(* IEC 61131-3 sources: s22-soft-shell/st_interpret/tests/test_inputs/execution/st_subset_8-9, 9 files *)

(* ---- counterinoutfunction.st ---- *)
// This function is designed to test IN_OUT variable.
// Takes in_out integer and adds 1 to it "counting up by 1"
// Then returns new count  with variable instead of function name
// function name returns true to indicate success
FUNCTION CounterInOutFunction : BOOL //BOOL is the return parameter data type
VAR_IN_OUT
  InOut1 :	INT; //IN_OUT parameter
END_VAR

  InOut1 := InOut1 + 1;

  CounterFunction:= 'TRUE'; //Set the return parameter

END_FUNCTION

(* ---- counteroutputfunction.st ---- *)
// This function is designed to test Output variable.
// Takes input integer and adds 1 to it "counting up by 1"
// Then returns new count using Output variable instead of function name
// function name returns true to indicate success
FUNCTION CounterOutputFunction : BOOL //BOOL is the return parameter data type
VAR_INPUT
  Input1 :	INT; //Input parameter
END_VAR
VAR_OUTPUT
  Output1 :	INT; //Output parameter
END_VAR

  Output1 := Input1 + 1;

  CounterFunction:= 'TRUE'; //Set the return parameter

END_FUNCTION

(* ---- simpleaddfunction.st ---- *)
FUNCTION SimpleAddFunction : INT //INT is the return parameter data type
VAR_INPUT
  Input1 :	INT; //Input parameter 1 to the function
  Input2 :	INT; //Input parameter 2 to the function
END_VAR

VAR
  Sum :	INT; //Local variable for temporary calculation
END_VAR

  Sum:= Input1 + Input2; //Total sum

  SimpleAddFunction:= Sum; //Set the return parameter

END_FUNCTION

(* ---- threevarfunction.st ---- *)
// This function is designed to test Output variable.
// Takes input integer and adds 1 to it "counting up by 1"
// Then returns new count using Output variable instead of function name
// function name returns true to indicate success
FUNCTION ThreeVarFunction : BOOL //BOOL is the return parameter data type
VAR_INPUT
  Input1 :	INT; //Input parameter
END_VAR
VAR_OUTPUT
  Output1 :	INT; //Output parameter
END_VAR
VAR_OUTPUT
  InOut1 :	INT; //Output parameter
END_VAR

  Output1 := Input1 + 1;

  InOut1  := InOut1 + 2;

  CounterFunction:= 'TRUE'; //Set the return parameter

END_FUNCTION

(* ---- valueaveragefunction.st ---- *)
FUNCTION ValueAverageFunction : REAL //REAL is the return parameter data type
VAR_INPUT
  Value1 :	REAL; //Input parameter 1 to the function
  Value2 :	REAL; //Input parameter 2 to the function
END_VAR

VAR
  Sum :	REAL; //Local variable for temporary calculation
END_VAR

  Sum:= Value1 + Value2; //Total sum
  Sum:= Sum/2; //Average

  ValueAverageFunction := Sum; //Set the return parameter

END_FUNCTION

(* ---- 09_Main_Add.st ---- *)
//Testing simple function call to add two numbers together
PROGRAM 09_Main_Add
    VAR
	a : int;
        b : int;
        result0 : int;
        result1 : int;
        result2 : int;
        result3 : int;
        ST_TESTING_RESULT : bool;
    END_VAR
        a := 3;
        b := 5;

        // four different ways of function input
        result0 := SimpleAddFunction(10, 10+5); // expects outputs of 25

        result1 := SimpleAddFunction(Input1 := 5, Input2 := 10);// expects outputs of 15

        result2 := SimpleAddFunction(a, b); // expects outputs of 8

        result3 := SimpleAddFunction(Input1 := a, Input2 := b); // expects outputs of 8

        ST_TESTING_RESULT := (result0 = 25 & result1 = 15) & (result2 = 8 & result3 = 8);

END_PROGRAM

(* ---- 09_Main_Avg.st ---- *)
//Testing simple function call to get average of two numbers
PROGRAM 09_Main_Avg
    VAR
	a : real;
        b : real;
        avg1 : real;
        avg2 : real;
        avg3 : real;
        avg4 : real;
        ST_TESTING_RESULT : bool;
    END_VAR
        a := 4;
        b := 6;

        // four different ways of function input
        avg1 := ValueAverageFunction(10, 10+5); // expects 12.5

        avg2 := ValueAverageFunction(Value1 := 5, Value2 := 10); // expects 7.5

        avg3 := ValueAverageFunction(a, b); // expects 5

        avg4 := ValueAverageFunction(Value1 := a, Value2 := b); // expects 5

        ST_TESTING_RESULT := (avg1 = 12.5 & avg2 = 7.5) & (avg3 = 5.0 & avg4 = 5.0);

END_PROGRAM

(* ---- 09_Main_Context_Check.st ---- *)
//Testing to insure seperation of context, Input2 and Sum variables being used in main and add function
PROGRAM 09_Main_Context_Check
    VAR
	    a : int;
        b : int;
        Input2 : int;
        Sum : INT;
        result0 : int;
        result1 : int;
        ST_TESTING_RESULT : bool;
    END_VAR
        a := 3;
        b := 5;
        Input2 := 10;
        Sum := 2;

        result0 := SimpleAddFunction(a, b); // expects outputs of 8

        result1 := SimpleAddFunction(Input1 := a, Input2 := b); // expects outputs of 8

        ST_TESTING_RESULT := (result0 = 8 & result1 = 8) & (Input2 = 10 & Sum = 2);

END_PROGRAM

(* ---- 09_Main_Demo_01.st ---- *)
// Testing for GO West Example use case example
// program doesnt go into while loop without C API
// is used to set INPUT1 or INPUT2 to TRUE
// x represents number of loops INPUT1 and INPUT2 are both true during
// OUTPUT1 represents number of loops
PROGRAM 09_Main_Demo_01
    VAR
	x : int;
        INPUT1 : bool;
        INPUT2 : bool;
        OUTPUT1 : int;
        ST_TESTING_RESULT : bool;
    END_VAR
        x := 0;
        INPUT1 := False;
        INPUT2 := False ;
        OUTPUT1 := 0 ;
//API would control INPUTs after here HERE here

        WHILE (INPUT1) OR (INPUT2) DO
            If (INPUT1) AND (INPUT2) THEN
                x:= x +1;
            END_IF;
            OUTPUT1 := SimpleAddFunction(Input1 := OUTPUT1, Input2 := 1);
        END_WHILE;
        ST_TESTING_RESULT := (x = 0 );
END_PROGRAM
